(* CoDeSys 2.3 export: VALUESENSORCLASS.EXP *)

(* Data type in ENUM *)
TYPE ValueSensorClass : (Differentiator:=1, Linearizator, StepSensor);
END_TYPE
